(* Schneider Machine Expert - Basic project automatic lamp control in warehouse, file version 2.7.0.0 *)
(* ProjectInformations: Name=New project *)

HARDWARE
  Cpu 0: TM221M16R/G
  EthernetConfiguration: NetworkName=M221, IpAllocationMode=FixedAddress, IpAddress=0.0.0.0, SubnetMask=0.0.0.0
  SerialLineConfiguration: Baud=Baud19200, Parity=ParityEven, DataBits=DataBits8, StopBits=StopBits1, PhysicalMedium=PhysicalMediumRs485, TransmissionMode=TransmissionModeModbusRtu, SlaveId=1, Addressing=SlaveAddressing
  MastTask: UsePeriodScanMode=false, PeriodScan=100
  FastTask: Period=255
  CpuBehavior: StartingMode=StartAsPreviousState, AutoSaveRamOnEeprom=true, WatchdogPeriod=250

SYMBOLS  (address, symbol, comment, settings)
  %I0.0     START_PB
  %I0.1     SWITCH1
  %I0.2     SWITCH2
  %I0.3     SWITCH3
  %I0.4     SWITCH4
  %I0.5     SWITCH5
  %I0.6     SWITCH6
  %I0.7     STOP
  %Q0.0     LAMP1
  %Q0.1     LAMP2
  %Q0.2     LAMP3
  %Q0.3     LAMP4
  %Q0.4     LAMP5
  %Q0.5     LAMP6
  %Q0.6     LAMP7
  %Q0.7     LMAP8

POU New POU
  (* SectionNumber=1 *)

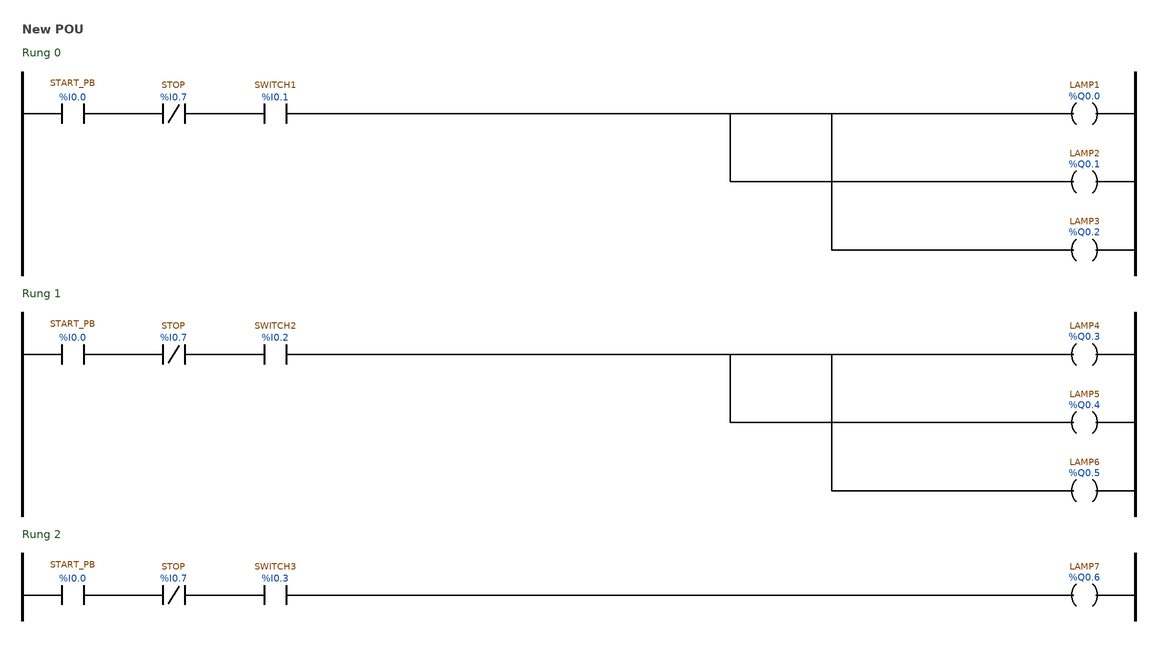

// Rung 0
  LD %I0.0                (* START_PB *)
  ANDN %I0.7              (* STOP *)
  AND %I0.1               (* SWITCH1 *)
  ST %Q0.0                (* LAMP1 *)
  ST %Q0.1                (* LAMP2 *)
  ST %Q0.2                (* LAMP3 *)
  // as ST:
  //   LAMP1 := START_PB AND NOT STOP AND SWITCH1;
  //   LAMP2 := START_PB AND NOT STOP AND SWITCH1;
  //   LAMP3 := START_PB AND NOT STOP AND SWITCH1;

// Rung 1
  LD %I0.0                (* START_PB *)
  ANDN %I0.7              (* STOP *)
  AND %I0.2               (* SWITCH2 *)
  ST %Q0.3                (* LAMP4 *)
  ST %Q0.4                (* LAMP5 *)
  ST %Q0.5                (* LAMP6 *)
  // as ST:
  //   LAMP4 := START_PB AND NOT STOP AND SWITCH2;
  //   LAMP5 := START_PB AND NOT STOP AND SWITCH2;
  //   LAMP6 := START_PB AND NOT STOP AND SWITCH2;

// Rung 2
  LD %I0.0                (* START_PB *)
  ANDN %I0.7              (* STOP *)
  AND %I0.3               (* SWITCH3 *)
  ST %Q0.6                (* LAMP7 *)
  // as ST:
  //   LAMP7 := START_PB AND NOT STOP AND SWITCH3;
